FUNCTION_BLOCK Test_AssertEquals_ULINT EXTENDS TUnitTestBase
VAR
    AssertionUnderTest : TAssertion(AssertionListenerMock);
    AssertionListenerMock : TAssertionListenerMock;
    ULINT_Variable : ULINT := 1111;
END_VAR

AssertionListenerMock.AssertionFailed  := FALSE;
AssertionListenerMock.AssertionMessage := '';
AssertionListenerMock.ExpectedAsString := '';
AssertionListenerMock.ActualAsString   := '';

// Test the assertion...
AssertionUnderTest.AssertEquals_ULINT(
    Expected := 2222,
    Actual   := ULINT_Variable,
    ObjectName := 'AssertionTest',
    VariableName := 'ULINT_Variable');
 
    
// Check the assertion worked...    
Assertion.AssertEquals_BOOL(
    Expected := TRUE,
    Actual   := AssertionListenerMock.AssertionFailed,
    ObjectName := _TestName,
    VariableName := 'AssertionListenerMock.AssertionFailed');

// Check the assertion messages...    
Assertion.AssertEquals_STRING(
    Expected := 'AssertEquals_ULINT failed in AssertionTest: Value "ULINT_Variable"',
    Actual   := AssertionListenerMock.AssertionMessage,
    ObjectName := _TestName,
    VariableName := 'AssertionListenerMock.AssertionMessage');

Assertion.AssertEquals_STRING(
    Expected := '  Expected = 2222',
    Actual   := AssertionListenerMock.ExpectedAsString,
    ObjectName := _TestName,
    VariableName := 'AssertionListenerMock.ExpectedAsString');

Assertion.AssertEquals_STRING(
    Expected := '  Actual   = 1111',
    Actual   := AssertionListenerMock.ActualAsString,
    ObjectName := _TestName,
    VariableName := 'AssertionListenerMock.ActualAsString');


TestFinished();

END_FUNCTION_BLOCK

(* stored: Version 1.1.0.1, ProductVersion 3.1.4024.3
   POU Test_AssertEquals_ULINT: Id {2d429d21-e8ad-4b9e-b6ce-98d13a034e5a}, SpecialFunc None *)
